FUNCTION_BLOCK AE_E_TO_EVENT (* Composite FB for convert AE to EVENT *)
  (* Standard: 61499-2; Description: Copyright (c) 2025 HR Agrartechnik GmbH This program and the accompanying materials are made available under the terms of the Eclipse Public License 2.0 which is available at https://www.eclipse.org/legal/epl-2.0/ SPDX-License-Identifier: EPL-2.0 *)
  (* Version 1.0, 2024-04-24, Franz Höpfinger, HR Agrartechnik GmbH *)
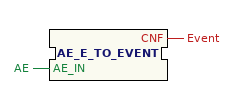
  EVENT_OUTPUT
    CNF; (* Confirmation from Adapter *)
  END_EVENT
  SOCKETS
    AE_IN : AE; (* Adapter Input *)
  END_SOCKETS
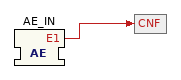
  EVENT_CONNECTIONS
    AE_IN.E1 TO CNF;
  END_CONNECTIONS
END_FUNCTION_BLOCK
